(* Schneider Machine Expert - Basic project partida_motores, file version 2.9.0.0 *)
(* ProjectInformations: Name=Novo projeto *)

HARDWARE
  Cpu 0: TM221CE24R
  EthernetConfiguration: NetworkName=M221, IpAllocationMode=FixedAddress, IpAddress=0.0.0.0, SubnetMask=0.0.0.0
  SerialLineConfiguration: Baud=Baud19200, Parity=ParityEven, DataBits=DataBits8, StopBits=StopBits1, PhysicalMedium=PhysicalMediumRs485, TransmissionMode=TransmissionModeModbusRtu, SlaveId=1, Addressing=SlaveAddressing
  MastTask: UsePeriodScanMode=false, PeriodScan=100
  FastTask: Period=255
  CpuBehavior: StartingMode=StartAsPreviousState, AutoSaveRamOnEeprom=true, WatchdogPeriod=250

SYMBOLS  (address, symbol, comment, settings)
  %M0       AUX_PAI_EMER_LIGA
  %M1       AUX_PAI_EMER_DESL
  %M2       AUX_PAI_LOCA
  %M3       AUX_PAI_REMO
  %M4       CMD_PAI_MOT1_LIGA
  %M5       CMD_PAI_MOT1_DESL
  %M6       CMD_PAI_MOT2_LIGA
  %M7       CMD_PAI_MOT2_DESL
  %M8       MOT1_LIGA_LOCAL
  %M9       MOT1_DESL_LOCAL
  %M10      MOT2_LIGA_LOCAL
  %M11      MOT2_DESL_LOCAL
  %M12      INI_REMO
  %M13      FIM_REMO
  %M50      HAB_MOT1
  %M51      HAB_MOT2
  %M100     CMD_IHM_INICIO
  %M101     CMD_IHM_FIM
  %I0.0     PAI_EMER
  %I0.1     PAI_LOCA
  %I0.2     PAI_REMO
  %I0.3     PAI_MOT1_LIGA
  %I0.4     PAI_MOT1_DESL
  %I0.5     PAI_MOT2_LIG
  %I0.6     PAI_MOT2_DESL

POU Novo POU
  (* SectionNumber=1 *)

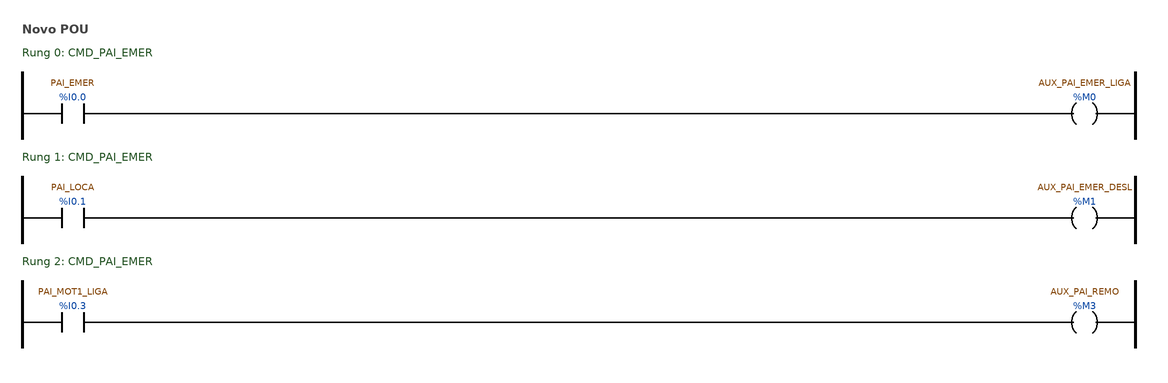

// Rung 0: CMD_PAI_EMER
  LD %I0.0                (* PAI_EMER *)
  ST %M0                  (* AUX_PAI_EMER_LIGA *)
  // as ST:
  //   AUX_PAI_EMER_LIGA := PAI_EMER;

// Rung 1: CMD_PAI_EMER
  LD %I0.1                (* PAI_LOCA *)
  ST %M1                  (* AUX_PAI_EMER_DESL *)
  // as ST:
  //   AUX_PAI_EMER_DESL := PAI_LOCA;

// Rung 2: CMD_PAI_EMER
  LD %I0.3                (* PAI_MOT1_LIGA *)
  ST %M3                  (* AUX_PAI_REMO *)
  // as ST:
  //   AUX_PAI_REMO := PAI_MOT1_LIGA;
